Staubli VAL3: setName.pgx

public program setName(string x_sName, num x_nIndex)
begin
  // set the name
  saveData:tData[x_nIndex].name=x_sName
end
